// TwinCAT 3 PLC project Plc
// ProgramVersion: 3.1.4024.0
// libraries:
//   Tc2_Standard, * (Beckhoff Automation GmbH)
//   Tc2_System, * (Beckhoff Automation GmbH)
//   Tc2_TcpIp, * (Beckhoff Automation GmbH)
//   Tc2_Utilities, * (Beckhoff Automation GmbH)
//   Tc3_Module, * (Beckhoff Automation GmbH)
// project tree:
//   Helper/ FN_MemoryClear.TcPOU
//   / PlcTask.TcTTO
//   POUs/ MAIN.TcPOU
//   POUs/TcpIp/ FB_TCP_IP_Server.TcPOU, FB_TCP_IP_ServerAccept.TcPOU, FB_TCP_IP_ServerClientConnection.TcPOU, FB_TCP_IP_SocketListen.TcPOU
// real-time tasks:
//   TASK PlcTask: cycle T#10ms, priority 20, ADS port 350

CONFIGURATION Plc
    RESOURCE PLC ON TwinCAT3
        TASK PlcTask(INTERVAL := T#10ms, PRIORITY := 20);
        PROGRAM MAIN WITH PlcTask : MAIN;
    END_RESOURCE
END_CONFIGURATION

// ---- POUs/MAIN.TcPOU
PROGRAM MAIN
VAR
	fbTCP_IP_Server: FB_TCP_IP_Server;
	fbTCP_IP_ServerClientConnection: FB_TCP_IP_ServerClientConnection;
END_VAR
VAR CONSTANT
END_VAR


fbTCP_IP_Server(
	sSrvNetId:= , 
	sLocalHost:= , 
	nLocalPort:= , 
	bListen:= , 
	bClose:= , 
	bReset:= , 
	TIMEOUT:= );

fbTCP_IP_ServerClientConnection();

END_PROGRAM

// ---- POUs/TcpIp/FB_TCP_IP_Server.TcPOU
FUNCTION_BLOCK FB_TCP_IP_Server
VAR_INPUT
	sSrvNetId: T_AmsNetId;
	sLocalHost: T_IPv4Addr := '192.168.1.7';
	nLocalPort: UDINT := 23;
	bListen: BOOL;
	bAccept: BOOL := TRUE;
	bClose: BOOL;
	bCloseAll: BOOL;
	bReset: BOOL;
	aSendDataBuffer: ARRAY[0..MAX_CLIENT] OF ARRAY[0..MAX_BUFFER] OF BYTE;		
	TIMEOUT: TIME := T#5S;	
END_VAR
VAR_OUTPUT
	aReceiveDataBuffer: ARRAY[0..MAX_CLIENT] OF ARRAY[0..MAX_BUFFER] OF BYTE;
	
END_VAR
VAR
	fbTCP_IP_SocketListen: FB_TCP_IP_SocketListen;
	fbSocketCloseAll: FB_SocketCloseAll;
	fbTCP_IP_ServerAccept: ARRAY[0..MAX_CLIENT] OF FB_TCP_IP_ServerAccept;
	bSend: ARRAY[0..MAX_CLIENT] OF BOOL;
	bClose2: ARRAY[0..MAX_CLIENT] OF BOOL;
	ftSocketListeningStopped: F_TRIG;
	i: INT;
	selection: INT := 0;
END_VAR
VAR CONSTANT
	MAX_BUFFER	: UINT:= 1023;
	MAX_CLIENT: UINT:= 2;
END_VAR


	ftSocketListeningStopped(CLK:= fbTCP_IP_SocketListen.bListening, Q=> );

	fbTCP_IP_SocketListen(
		sSrvNetId			:= sSrvNetId, 
		sLocalHost			:= sLocalHost, 
		nLocalPort			:= nLocalPort, 
		bListen				:= bListen, 
		bClose				:= bClose, 
		bReset				:= bReset, 
		TIMEOUT				:= TIMEOUT, 
		bDone				=> , 
		bBusy				=> , 
		bListening			=> , 
		hListener			=> , 
		bError				=> , 
		nErrID				=> , 
		sStatus				=> );	
		
	FOR i := 0 TO MAX_CLIENT BY 1 DO
		fbTCP_IP_ServerAccept[i](
			sSrvNetId			:= sSrvNetId, 
			bAccept				:= bAccept, 
			bListenReady		:= fbTCP_IP_SocketListen.bListening, 
			hListener			:= fbTCP_IP_SocketListen.hListener, 
			bSend				:= bSend[i], 
			bClose				:= bClose2[i] OR ftSocketListeningStopped.Q, 
			bReset				:= bReset, 
			aSendDataBuffer		:= aSendDataBuffer[i], 
			TIMEOUT				:= TIMEOUT, 
			bAccepted			=> , 
			bError				=> , 
			nErrID				=> , 
			sStatus				=> , 
			aReceiveDataBuffer	=> aReceiveDataBuffer[i]);			
	END_FOR

	selection;
	fbTCP_IP_ServerAccept[0].bAccepted;
	fbTCP_IP_ServerAccept[1].bAccepted;
	fbTCP_IP_ServerAccept[2].bAccepted;
	fbTCP_IP_ServerAccept[selection].bError;
	fbTCP_IP_ServerAccept[selection].nErrID;
	fbTCP_IP_ServerAccept[selection].sStatus;
	aReceiveDataBuffer[0][0];
	aReceiveDataBuffer[0][1];
	aReceiveDataBuffer[0][2];
	aReceiveDataBuffer[0][3];

	aReceiveDataBuffer[1][0];
	aReceiveDataBuffer[1][1];
	aReceiveDataBuffer[1][2];
	aReceiveDataBuffer[1][3];

	aReceiveDataBuffer[2][0];
	aReceiveDataBuffer[2][1];
	aReceiveDataBuffer[2][2];
	aReceiveDataBuffer[2][3];
	
		
	fbSocketCloseAll(
		sSrvNetId			:= sSrvNetId, 
		bExecute			:= bCloseAll, 
		tTimeout			:= T#5S, 
		bBusy				=> , 
		bError				=> , 
		nErrId				=> );

END_FUNCTION_BLOCK

// ---- POUs/TcpIp/FB_TCP_IP_SocketListen.TcPOU
FUNCTION_BLOCK FB_TCP_IP_SocketListen
VAR_INPUT
	sSrvNetId: T_AmsNetId;
	sLocalHost: T_IPv4Addr;
	nLocalPort: UDINT;
	bListen: BOOL;		//	1: Listen | 0: Stop listening, remove all existing connections
	bClose: BOOL;
	bReset: BOOL;
	TIMEOUT: TIME := T#5s;
	
END_VAR
VAR_OUTPUT
	bDone: BOOL;
	bBusy: BOOL;
	bListening: BOOL;
	hListener: Tc2_TcpIp.T_HSOCKET;
	bError: BOOL;
	nErrID: UDINT;
	sStatus: STRING(255);
	
END_VAR
VAR
	step: (eInit, eInitToListen, eListen, eWait, eClose, eClose2, eError);
	fbSocketListen: FB_SocketListen;
	fbSocketClose: FB_SocketClose;
	
	tonCaseStuck: TON;
	rtClose: R_TRIG;
	M_Close: BOOL;
	tonCloseCmdOverride: TON;
	rtReset: R_TRIG;
	M_Reset: BOOL;
	tonResetCmdOverride: TON;
	tonAutoErrorReset: TON;
	_doneSetFromCloseCase: BOOL;
	_doneSetFromListenCase: BOOL;
END_VAR

	
	rtClose(CLK:= bClose, Q=> );
	IF rtClose.Q THEN
		M_Close			:=	TRUE;
	END_IF
	tonCloseCmdOverride(IN:= M_Close, PT:= TIMEOUT + T#1S, Q=> , ET=> );
	IF tonCloseCmdOverride.Q THEN
		step		:=	eClose;
		M_Close		:=	FALSE;			
	END_IF

	rtReset(CLK:= bReset, Q=> );
	IF rtReset.Q THEN
		M_Reset			:=	TRUE;
	END_IF
	
	IF bDone AND tonResetCmdOverride.Q THEN
		step		:=	eInit;
		M_Reset		:=	FALSE;
		bDone		:=	FALSE;	
	END_IF
	tonResetCmdOverride(IN:= M_Reset, PT:= TIMEOUT + T#1S, Q=> , ET=> );
	IF tonResetCmdOverride.Q THEN
		bDone		:=	TRUE;		
	END_IF
	
	CASE step OF
	eInit:
		IF M_Close AND (NOT bReset) THEN
			step		:=	eClose;
			M_Close		:=	FALSE;
			bBusy		:=	TRUE;
			bDone		:=	FALSE;
		ELSIF bListen AND (NOT bReset) AND (NOT bClose) THEN
			step		:=	eInitToListen;		
			fbSocketListen(bExecute:= FALSE);
			fbSocketClose(bExecute:=	FALSE);
			bListening	:=	FALSE;
			bBusy		:=	TRUE;
			bDone		:=	FALSE;
		END_IF
		M_Reset			:=	FALSE;
		tonAutoErrorReset(IN:= FALSE);
		tonCaseStuck(IN:= FALSE);
		
		IF _doneSetFromCloseCase AND bDone AND NOT bClose THEN
			_doneSetFromCloseCase	:=	FALSE;
			bDone					:=	FALSE;
		END_IF
		
	eInitToListen:
		tonCaseStuck(IN:= TRUE, PT:= TIMEOUT + T#2S, Q=> , ET=> );

		fbSocketListen(
			sSrvNetId		:= sSrvNetId, 
			sLocalHost		:= sLocalHost, 
			nLocalPort		:= nLocalPort, 
			bExecute		:= TRUE, 
			tTimeout		:= TIMEOUT, 
			bBusy			=> , 
			bError			=> , 
			nErrId			=> , 
			hListener		=> hListener);		
		
		IF fbSocketListen.bError THEN
			step		:=	eError;
			nErrID		:=	fbSocketListen.nErrId;
			sStatus		:=	'FB Error: fbSocketListen | case no. eInitToListen';			
		ELSIF (fbSocketListen.bBusy) THEN
			step		:=	eListen;
			tonCaseStuck(IN:= FALSE);	
		END_IF
		
		IF tonCaseStuck.Q THEN
			IF M_Close THEN				
				step		:=	eClose;
				M_Close		:=	FALSE;
				tonCaseStuck(IN:= FALSE);
			ELSE
				step		:=	eError;
				nErrID		:=	1;
				sStatus		:=	'Custom ErrID | Case stuck: eInitToListen';
				tonCaseStuck(IN:= FALSE);	
			END_IF
		END_IF
		
	eListen:
		tonCaseStuck(IN:= TRUE, PT:= TIMEOUT + T#2S, Q=> , ET=> );

		fbSocketListen(
			sSrvNetId		:= sSrvNetId, 
			sLocalHost		:= sLocalHost, 
			nLocalPort		:= nLocalPort, 
			bExecute		:= TRUE, 
			tTimeout		:= TIMEOUT, 
			bBusy			=> , 
			bError			=> , 
			nErrId			=> , 
			hListener		=> hListener);		
		
		IF fbSocketListen.bError THEN
			step		:=	eError;
			nErrID		:=	fbSocketListen.nErrId;
			sStatus		:=	'FB Error: fbSocketListen | case no. eListen';			
		ELSIF (NOT fbSocketListen.bBusy) THEN
			fbSocketListen(bExecute:= FALSE);
			IF M_Close THEN
				step		:=	eClose;
				M_Close		:=	FALSE;
				tonCaseStuck(IN:= FALSE);
			ELSE
				step		:=	eWait;
				bListening	:=	TRUE;
				bBusy		:=	FALSE;
				bDone		:=	TRUE;
				_doneSetFromListenCase	:=	TRUE;
				tonCaseStuck(IN:= FALSE);
				bError		:=	FALSE;
				nErrID		:=	0;
				sStatus		:=	'';
			END_IF
		END_IF	

		IF tonCaseStuck.Q THEN
			IF M_Close THEN				
				step		:=	eClose;
				M_Close		:=	FALSE;
				tonCaseStuck(IN:= FALSE);
			ELSE
				step		:=	eError;
				nErrID		:=	1;
				sStatus		:=	'Custom ErrID | Case stuck: eListen';
				tonCaseStuck(IN:= FALSE);	
			END_IF				
		END_IF
		
	eWait:
		IF NOT bListen THEN
			step		:=	eClose;
			bDone		:=	FALSE;
			_doneSetFromListenCase	:=	FALSE;
		ELSIF M_Close THEN
			step		:=	eClose;	
			M_Close		:=	FALSE;
			bDone		:=	FALSE;
			_doneSetFromListenCase	:=	FALSE;
		ELSIF M_Reset THEN
			step		:=	eInit;
			bListening	:=	FALSE;
			M_Reset		:=	FALSE;
			bDone		:=	FALSE;
			_doneSetFromListenCase	:=	FALSE;	
		END_IF

		
	eClose:
		tonCaseStuck(IN:= TRUE, PT:= TIMEOUT + T#2S, Q=> , ET=> );

		bListening	:=	FALSE;
		M_Close		:=	FALSE;
		
		fbSocketClose(
			sSrvNetId		:= sSrvNetId, 
			hSocket			:= fbSocketListen.hListener, 
			bExecute		:= TRUE, 
			tTimeout		:= TIMEOUT, 
			bBusy			=> , 
			bError			=> , 
			nErrId			=> );
			
		IF fbSocketClose.bError THEN
			step		:=	eError;
			nErrID		:=	fbSocketClose.nErrId;
			sStatus		:=	'FB Error: fbSocketClose | case no. eClose';			
		ELSIF (NOT fbSocketClose.bBusy) THEN
			step		:=	eClose2;
			tonCaseStuck(IN:= FALSE);
		END_IF	
		
		IF tonCaseStuck.Q THEN
			step		:=	eError;
			nErrID		:=	1;
			sStatus		:=	'Custom ErrID | Case stuck: eClose';
			tonCaseStuck(IN:= FALSE);	
		END_IF
	
	eClose2:
		tonCaseStuck(IN:= TRUE, PT:= TIMEOUT + T#2S, Q=> , ET=> );

		fbSocketClose(
			sSrvNetId		:= sSrvNetId, 
			hSocket			:= fbSocketListen.hListener, 
			bExecute		:= TRUE, 
			tTimeout		:= TIMEOUT, 
			bBusy			=> , 
			bError			=> , 
			nErrId			=> );
			
		IF fbSocketClose.bError THEN
			step		:=	eError;
			nErrID		:=	fbSocketClose.nErrId;
			sStatus		:=	'FB Error: fbSocketClose | case no. eClose';			
		ELSIF (NOT fbSocketClose.bBusy) THEN
			fbSocketClose(bExecute:= FALSE);
			step		:=	eInit;
			bBusy		:=	FALSE;
			bDone		:=	TRUE;
			_doneSetFromCloseCase	:=	TRUE;
			tonCaseStuck(IN:= FALSE);
		END_IF	
		
		IF tonCaseStuck.Q THEN
			step		:=	eError;
			nErrID		:=	1;
			sStatus		:=	'Custom ErrID | Case stuck: eClose';
			tonCaseStuck(IN:= FALSE);	
		END_IF		
			
	eError:
		bError		:=	TRUE;
		bBusy		:=	FALSE;
		bDone		:=	FALSE;
		
		bListening	:=	FALSE;
		fbSocketListen(bExecute:= FALSE);
		fbSocketClose(bExecute:= FALSE);
		tonCaseStuck(IN:= FALSE);
		
		tonAutoErrorReset(IN:= bListen, PT:= T#5S, Q=> , ET=> );
		IF tonAutoErrorReset.Q THEN
			step	:=	eInit;
			tonAutoErrorReset(IN:= FALSE);
			
		END_IF
		
		IF M_Close THEN
			step	:=	eClose;
			M_Close	:=	FALSE;
			tonAutoErrorReset(IN:= FALSE);
			bError		:=	FALSE;
			nErrID		:=	0;
			sStatus		:=	'';
		ELSIF M_Reset THEN
			step	:=	eInit;
			M_Reset	:=	FALSE;
			tonAutoErrorReset(IN:= FALSE);
			bError		:=	FALSE;
			nErrID		:=	0;
			sStatus		:=	'';	
		END_IF
		
	END_CASE
	

	
	
	//	Calling
	fbSocketListen();
	fbSocketClose();
	tonCaseStuck();
	tonAutoErrorReset();

END_FUNCTION_BLOCK

// ---- POUs/TcpIp/FB_TCP_IP_ServerAccept.TcPOU
FUNCTION_BLOCK FB_TCP_IP_ServerAccept
VAR_INPUT
	sSrvNetId: T_AmsNetId;
	bAccept: BOOL;
	bListenReady: BOOL;
	hListener: Tc2_TcpIp.T_HSOCKET;
	bSend: BOOL;
	bClose: BOOL;
	bReset: BOOL;
	aSendDataBuffer: ARRAY[0..MAX_BUFFER] OF BYTE;	
	TIMEOUT: TIME := T#5S;
	
END_VAR
VAR_OUTPUT
	//bDone: BOOL;
	//bBusy: BOOL;
	bAccepted: BOOL;
	bError: BOOL;
	nErrID: UDINT;
	sStatus: STRING(255);
	aReceiveDataBuffer: ARRAY[0..MAX_BUFFER] OF BYTE;
END_VAR
VAR
	step: (eInit, ePreAccept, eAccept, eManageConnection, eWait, ePreSend, eSend, eClose, eClose2, eCloseAll, eError);
	fbSocketAccept: FB_SocketAccept;
	fbSocketClose: FB_SocketClose;
	fbSocketSend: FB_SocketSend;
	fbSocketReceive: FB_SocketReceive;
	aDataBuffer: ARRAY[0..MAX_BUFFER] OF BYTE;
	nRecBytes: UDINT;

	rtSend: R_TRIG;
	rtClose: R_TRIG;
	tonReceivePollFreq: TON;
	rtReset: R_TRIG;
	tonError: TON;
	
	M_Close: BOOL;
	tonCloseCmdOverride: TON;
	M_Reset: BOOL;
	tonResetCmdOverride: TON;
	//tonCaseStuck: TON;
	tonAutoErrorReset: TON;
	nBytesTransferred: UDINT;
END_VAR
VAR CONSTANT
	MAX_BUFFER	: UINT:= 1023;
END_VAR

	rtClose(CLK:= bClose, Q=> );
	IF rtClose.Q THEN
		M_Close			:=	TRUE;
	END_IF
	tonCloseCmdOverride(IN:= M_Close, PT:= TIMEOUT + T#1S, Q=> , ET=> );
	IF tonCloseCmdOverride.Q THEN
		step		:=	eClose;
		M_Close		:=	FALSE;			
	END_IF

	rtReset(CLK:= bReset, Q=> );
	IF rtReset.Q THEN
		M_Reset			:=	TRUE;
	END_IF
	
//	IF bDone AND tonResetCmdOverride.Q THEN
//		step		:=	eInit;
//		M_Reset		:=	FALSE;
//		bDone		:=	FALSE;	
//	END_IF
	tonResetCmdOverride(IN:= M_Reset, PT:= TIMEOUT + T#1S, Q=> , ET=> );
	IF tonResetCmdOverride.Q THEN
		//bDone		:=	TRUE;	
		step		:=	eInit;
		M_Reset		:=	FALSE;	
	END_IF

	CASE step OF
	eInit:
		IF bAccept AND (bListenReady AND hListener.handle <> 0) AND (NOT bReset) AND (NOT bClose) THEN
			step		:=	ePreAccept;
			bAccepted	:=	FALSE;
		ELSIF M_Close AND (NOT bReset) THEN
			step		:=	eClose;
			M_Close		:=	FALSE;
		END_IF
		fbSocketAccept(bExecute:= FALSE);
		fbSocketClose(bExecute:= FALSE);
		fbSocketSend(bExecute:= FALSE);
		M_Reset			:=	FALSE;
		
	ePreAccept:
		fbSocketAccept(
			sSrvNetId		:= sSrvNetId, 
			hListener		:= hListener, 
			bExecute		:= TRUE, 
			tTimeout		:= TIMEOUT, 
			bAccepted		=> , 
			bBusy			=> , 
			bError			=> , 
			nErrId			=> , 
			hSocket			=> );
	
		IF fbSocketAccept.bError THEN
			step		:=	eError;
			nErrID		:=	fbSocketAccept.nErrId;
			sStatus		:=	'FB Error: fbSocketAccept | case no. ePreAccept';
		ELSE			
		//ELSIF (fbSocketAccept.bBusy) THEN	- Note: Observed that this FB does not trigger Busy bit
			step		:=	eAccept;
		END_IF

	eAccept:
		fbSocketAccept(
			sSrvNetId		:= sSrvNetId, 
			hListener		:= hListener, 
			bExecute		:= TRUE, 
			tTimeout		:= TIMEOUT, 
			bAccepted		=> , 
			bBusy			=> , 
			bError			=> , 
			nErrId			=> , 
			hSocket			=> );
			
		IF fbSocketAccept.bError THEN
			step		:=	eError;
			nErrID		:=	fbSocketAccept.nErrId;
			sStatus		:=	'FB Error: fbSocketAccept | case no. eAccept';
		ELSIF (NOT fbSocketAccept.bBusy) THEN
			IF fbSocketAccept.hSocket.handle <> 0 THEN
				step			:=	eManageConnection;
				bAccepted		:=	fbSocketAccept.bAccepted;
			ELSE
				step			:=	eManageConnection;
			END_IF	
			bError		:=	FALSE;
			nErrID		:=	0;
			sStatus		:=	'';
		END_IF	

	eManageConnection:
		IF NOT bAccepted THEN
			step		:=	eInit;
		ELSE
			step		:=	eWait;
		END_IF
	
	eWait:	
		IF rtSend.Q THEN
			step		:=	ePreSend;
		END_IF
		IF M_Close THEN
			M_Close		:=	FALSE;
			step		:=	eClose;
		END_IF
	
	ePreSend:
		fbSocketSend(
			sSrvNetId		:= sSrvNetId, 
			hSocket			:= fbSocketAccept.hSocket, 
			cbLen			:= SIZEOF(aSendDataBuffer), 
			pSrc			:= ADR(aSendDataBuffer), 
			bExecute		:= TRUE, 
			tTimeout		:= TIMEOUT, 
			bBusy			=> , 
			bError			=> , 
			nErrId			=> );	
	
		IF fbSocketSend.bError THEN
			step			:=	eError;
			nErrID			:=	fbSocketSend.nErrId;
			sStatus			:=	'FB_SocketSend | error case: ePreSend';
		ELSIF (fbSocketSend.bBusy) THEN
			fbSocketSend(bExecute	:=	FALSE);
			step			:=	eSend;		
		END_IF			
		
	eSend:
		fbSocketSend(
			sSrvNetId		:= sSrvNetId, 
			hSocket			:= fbSocketAccept.hSocket, 
			cbLen			:= SIZEOF(aSendDataBuffer), 
			pSrc			:= ADR(aSendDataBuffer), 
			bExecute		:= TRUE, 
			tTimeout		:= TIMEOUT, 
			bBusy			=> , 
			bError			=> , 
			nErrId			=> );	
	
		IF fbSocketSend.bError THEN
			step			:=	eError;
			nErrID			:=	fbSocketSend.nErrId;
			sStatus			:=	'FB_SocketSend | error case: eSend';
		ELSIF (NOT fbSocketSend.bBusy) THEN
			fbSocketSend(bExecute	:=	FALSE);
			step			:=	eWait;		
		END_IF	
		
	eClose:		
		bAccepted			:=	FALSE;
		
		fbSocketClose(
			sSrvNetId		:= sSrvNetId, 
			hSocket			:= fbSocketAccept.hSocket, 
			bExecute		:= TRUE, 
			tTimeout		:= TIMEOUT, 
			bBusy			=> , 
			bError			=> , 
			nErrId			=> );
			
		IF fbSocketClose.bError THEN
			step		:=	eError;
			nErrID		:=	fbSocketClose.nErrId;
			sStatus		:=	'FB Error: fbSocketClose | case no. eClose';			
		ELSIF (NOT fbSocketClose.bBusy) THEN
			step		:=	eClose2;
		END_IF	
	
	eClose2:

		fbSocketClose(
			sSrvNetId		:= sSrvNetId, 
			hSocket			:= fbSocketAccept.hListener, 
			bExecute		:= TRUE, 
			tTimeout		:= TIMEOUT, 
			bBusy			=> , 
			bError			=> , 
			nErrId			=> );
			
		IF fbSocketClose.bError THEN
			step		:=	eError;
			nErrID		:=	fbSocketClose.nErrId;
			sStatus		:=	'FB Error: fbSocketClose | case no. eClose';			
		ELSIF (NOT fbSocketClose.bBusy) THEN
			fbSocketClose(bExecute:= FALSE);
			step		:=	eInit;

		END_IF	
		
	eError:
		bError		:=	TRUE;
		//bBusy		:=	FALSE;
		//bDone		:=	FALSE;
		
		bAccepted	:=	FALSE;
		fbSocketAccept(bExecute:= FALSE);
		fbSocketClose(bExecute:= FALSE);
		fbSocketSend(bExecute:= FALSE);
		
		tonAutoErrorReset(IN:= bAccept, PT:= T#5S, Q=> , ET=> );
		IF tonAutoErrorReset.Q THEN
			step	:=	eInit;
			tonAutoErrorReset(IN:= FALSE);			
		END_IF
		
		IF M_Close THEN
			step	:=	eClose;
			M_Close	:=	FALSE;
			tonAutoErrorReset(IN:= FALSE);
			bError		:=	FALSE;
			nErrID		:=	0;
			sStatus		:=	'';
		ELSIF M_Reset THEN
			step	:=	eInit;
			M_Reset	:=	FALSE;
			tonAutoErrorReset(IN:= FALSE);
			bError		:=	FALSE;
			nErrID		:=	0;
			sStatus		:=	'';	
		END_IF
		
	END_CASE
	
	tonReceivePollFreq(IN:= (NOT tonReceivePollFreq.Q) AND 
							bAccepted AND 
							(NOT bError) AND 
							(NOT fbSocketReceive.bBusy), 
						PT:= T#1S, Q=> , ET=> );
	
		fbSocketReceive(
			sSrvNetId		:= sSrvNetId, 
			hSocket			:= fbSocketAccept.hSocket, 
			cbLen			:= SIZEOF(aDataBuffer), 
			pDest			:= ADR(aDataBuffer), 
			bExecute		:= tonReceivePollFreq.Q, 
			tTimeout		:= TIMEOUT, 
			bBusy			=> , 
			bError			=> , 
			nErrId			=> , 
			nRecBytes		=> nRecBytes);	
		
		IF fbSocketReceive.nRecBytes > 0 THEN			
			FN_MemoryClear(destAddr:= ADR(aReceiveDataBuffer), Len:= SIZEOF(aReceiveDataBuffer));
		
			nBytesTransferred	:=	MEMCPY(destAddr:= ADR(aReceiveDataBuffer), srcAddr:= ADR(aDataBuffer), n:= nRecBytes);
			IF (nRecBytes <> nBytesTransferred) AND step = eWait THEN
				bError		:=	TRUE;
				nErrID		:=	1;
				sStatus		:=	'Bytes transfered is nt equal to received bytes | Custom Error ID';
				step		:=	eError;
			END_IF
		END_IF

END_FUNCTION_BLOCK

// ---- Helper/FN_MemoryClear.TcPOU
FUNCTION FN_MemoryClear
VAR_INPUT
	destAddr: PVOID;
	Len: UDINT;
END_VAR
VAR
	NULL: BYTE:= 0;
	i: ULINT;
END_VAR


	FOR i := 0 TO (Len-1) BY 1 DO
		MEMCPY(destAddr:= destAddr + i, srcAddr:= ADR(NULL), n:= 1);				
	END_FOR

END_FUNCTION

// ---- POUs/TcpIp/FB_TCP_IP_ServerClientConnection.TcPOU
FUNCTION_BLOCK FB_TCP_IP_ServerClientConnection
VAR_INPUT
	sSrvNetId: T_AmsNetId;
	sLocalHost: T_IPv4Addr := '192.168.1.7';
	nLocalPort: UDINT := 23;
	
END_VAR
VAR_OUTPUT
	
END_VAR
VAR
	fbServerClientConnection: FB_ServerClientConnection;
	hServer: T_HSERVER;
	eMode: E_SocketAcceptMode;
	sRemoteHost: T_IPv4Addr := '192.168.1.7';
	nRemotePort: UDINT := 23;
	bEnable: BOOL;
	tReconnect: TIME := T#2s;
	bEnable2: BOOL;
END_VAR


	F_CreateServerHnd(
		sSrvNetID			:= sSrvNetID, 
		sLocalHost			:= sLocalHost, 
		nLocalPort			:= nLocalPort, 
		nMode				:= LISTEN_MODE_CLOSEALL, 
		bEnable				:= bEnable2, 
		hServer				:= hServer);

	fbServerClientConnection(
		hServer				:= hServer, 
		eMode				:= eMode, 
		sRemoteHost			:= sRemoteHost, 
		nRemotePort			:= nRemotePort, 
		bEnable				:= bEnable, 
		tReconnect			:= tReconnect, 
		bBusy				=> , 
		bError				=> , 
		nErrID				=> , 
		hSocket				=> , 
		eState				=> );

	fbServerClientConnection.bBusy;
	fbServerClientConnection.bError;
	fbServerClientConnection.nErrID;
	fbServerClientConnection.hSocket.handle;
	fbServerClientConnection.eState;

END_FUNCTION_BLOCK
